// TIA Portal V18 export
TYPE "UDT_IAI_Axis_Positions"
// =================================================================================
//  POSITION SETS - Mirroring the Axis Driver's Position Array
//  =================================================================================
   STRUCT
      Position { S7_SetPoint := 'True'} : Array[1..20] of "UDT_Motion_Point_IAI";
   END_STRUCT;
END_TYPE
